RoboDK station: Solution.rdk

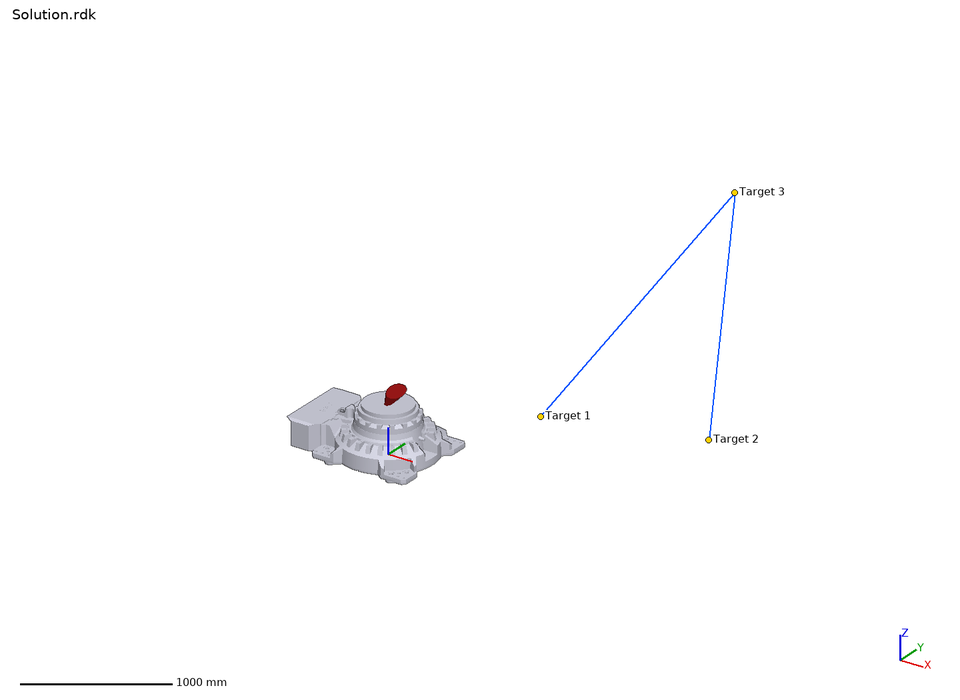
[picture v0: the station drawn from its stored meshes, robots at their saved joint values, targets as dots, program paths as lines]
Station Project_Q3 (saved by RoboDK 5.4.3). Poses are relative to the parent item; angles as X-Y-Z fixed-axis rotations.
  - frame ABB IRB 6700-150/3.20 Base at (0, 0, 0) mm
    - robot ABB IRB 6700-150/3.20: 6 axes, payload 150 kg, reach 3200 mm, repeatability 0.06 mm, weight 1280 kg
        joint limits [-170, -65, -180, -300, -130, -360] to [170, 85, 70, 300, 130, 360]; home [0, 0, 0, 0, 0, 0]; saved at [-16.89, 37.06, -19, -57.62, -12.91, 12.94]
      - tool Generic Paint Sprayer, TCP at (50, 0, 450) mm, rotated rx 0 ry 30 rz 0 deg, size 203.2 x 279.7 x 471.5 mm
    - target Target 1 (Cartesian target) at (2555.46, -1903.96, 1750.76) mm, rotated rx -120.65 ry 37.03 rz -159.14 deg; joints [-38.28, 28.99, -19, -57.62, -12.91, 12.94] of ABB IRB 6700-150/3.20
    - target Target 2 (Cartesian target) at (3177.09, -872.15, 1338.87) mm, rotated rx -128.87 ry 32.6 rz -142.46 deg; joints [-16.89, 37.06, -19, -57.62, -12.91, 12.94] of ABB IRB 6700-150/3.20
    - target Target 3 (Cartesian target) at (2713.69, 88.53, 2630.38) mm, rotated rx -97.53 ry 44.65 rz -105.59 deg; joints [0, 10, -19, -57.62, -12.91, 12.94] of ABB IRB 6700-150/3.20
  - program Prog1 (5 instructions, listed below)
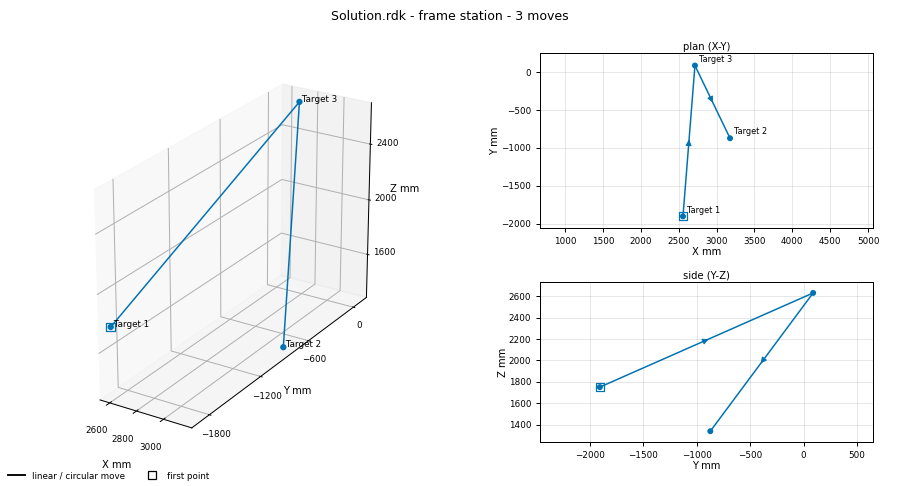
[picture p0: tool path of Solution.rdk in frame station, 3 of 3 moves have a stored position in this frame; points joined in program order, loops and branches not executed]

--- program Prog1 (robot ABB IRB 6700-150/3.20) ---
  Set Ref.: ABB IRB 6700-150/3.20 Base
  Set Tool: Generic Paint Sprayer
  MoveJ (Target 1)
  MoveL (Target 3)
  MoveL (Target 2)
